// TIA Portal V17 export
// export: Created 2022-07-16T16:56:14.3916578Z, ExportSetting WithDefaults, DisplayName Totally Integrated Automation Portal, DisplayVersion V17, DisplayName TIA Portal Openness, DisplayVersion V17, DisplayName TIA Portal Version Control Interface, DisplayVersion V17, DisplayName TIA Portal Test Suite Advanced, DisplayVersion V17, DisplayName STEP 7 Professional, DisplayVersion V17, DisplayName STEP 7 Safety, DisplayVersion V17, DisplayName WinCC Professional, DisplayVersion V17
TYPE "Client interface_1.dbData.postTestResult.mainSequence.pressure"
// stored: IsFailsafeCompliant false
   STRUCT
      postPressurizationPeriod { ExternalWritable := 'False'} : Bool;
      postDwellPeriod { ExternalWritable := 'False'} : Bool;
      bleedInterval1 { ExternalWritable := 'False'} : Bool;
      bleedInterval2 { ExternalWritable := 'False'} : Bool;
      bleedInterval3 { ExternalWritable := 'False'} : Bool;
      bleedInterval4 { ExternalWritable := 'False'} : Bool;
      bleedInterval5 { ExternalWritable := 'False'} : Bool;
      bleedInterval6 { ExternalWritable := 'False'} : Bool;
      bleedInterval7 { ExternalWritable := 'False'} : Bool;
      bleedInterval8 { ExternalWritable := 'False'} : Bool;
      bleedInterval9 { ExternalWritable := 'False'} : Bool;
      bleedInterval10 { ExternalWritable := 'False'} : Bool;
      bleedInterval11 { ExternalWritable := 'False'} : Bool;
      bleedInterval12 { ExternalWritable := 'False'} : Bool;
      mechanicalFailsavePressure { ExternalWritable := 'False'} : Bool;
   END_STRUCT;
END_TYPE
